// This function has been automatically generated from the project information.
{attribute 'signature_flag' := '1073741824'}
{attribute 'TcGenerated'}
{attribute 'no-analysis'}
FUNCTION F_GetTitle : WSTRING
VAR_INPUT
	
END_VAR

F_GetTitle := "CNM AoC Lib";

END_FUNCTION

(* stored: Version 1.1.0.1
   POU F_GetTitle: Id {d05f4c71-73f3-4953-903d-5434c3eea964}, SpecialFunc None *)
